Fanuc KAREL source: ka00225.KL

-- PROVISIONAL review KL for V770-1; original PC SHA256 a7dc76903850cb91fe79d1eecedecd5ba942976ea1eb5713bf1ff352b2a7d014
-- Incomplete behavior may be omitted. Consult companion uncertainty JSON. Do not deploy.
PROGRAM KA00225
%NOLOCKGROUP
BEGIN
  -- UNRESOLVED_PC offsets 5-19; opcodes 22,22,1E
  -- UNRESOLVED_PC offsets 24-28; opcodes 7F
END KA00225
